FUNCTION_BLOCK FB_RingBuffer
VAR
END_VAR

END_FUNCTION_BLOCK

(* stored: Version 1.1.0.1
   POU FB_RingBuffer: Id {33c9426c-7440-438e-b718-b6fa38b9b4e1}, SpecialFunc None *)
